// TwinCAT 3 PLC project PLC1
// ProgramVersion: 3.1.4024.0
// libraries:
//   Tc2_Standard, * (Beckhoff Automation GmbH)
//   Tc2_System, * (Beckhoff Automation GmbH)
//   Tc3_Module, * (Beckhoff Automation GmbH)
//   VisuSymbols,3.5.10.0,System
// project tree:
//   / Gestore di visualizzazione.TcVMO (not stored), GlobalTextList.TcGTLO, PlcTask.TcTTO (not stored)
//   GVLs/ GVL.TcGVL (not stored)
//   POUs/ MAIN.TcPOU
//   VISUs/ Screen1.TcVIS (not stored)

// ---- POUs/MAIN.TcPOU
PROGRAM MAIN
VAR
END_VAR

MarciaArrestoMotore();

ACTION MarciaArrestoMotore:
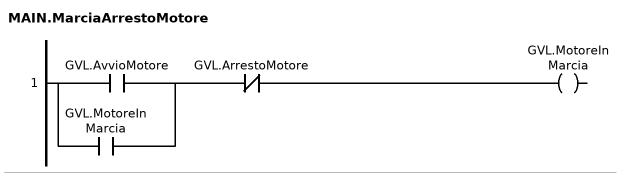
// NETWORK 1
GVL.MotoreInMarcia := (GVL.AvvioMotore OR GVL.MotoreInMarcia) AND NOT GVL.ArrestoMotore;
END_ACTION

END_PROGRAM

// ---- GlobalTextList.TcGTLO
TEXTLIST GlobalTextList
  88 = 'Arresto'
  599 = 'Marcia'
  849 = 'Motor'
  673 = 'Motore'
  613 = 'Screen 1'
  286 = 'Start'
  74 = 'Stop'
END_TEXTLIST
